(* IEC 61131-3 sources: Industry-PLC-LLM/data/PLCBEAD_repo/PLCBEAD_PLCEmbed-main/PLC-BEAD/Source/GEB/HYST_3, 1 file *)

(* ---- HYST_3.ST ---- *)
FUNCTION_BLOCK HYST_3_Block

	VAR_INPUT
		IN :	REAL;
		HYST :	REAL;
		VAL1 :	REAL;
		VAL2 :	REAL;
	END_VAR

	VAR_OUTPUT
		Q1 :	BOOL;
		Q2 :	BOOL;
	END_VAR

	VAR
		X :	REAL;
	END_VAR

	X := HYST * 0.5;
	IF IN < VAL1 - X THEN
		Q1 := TRUE;
	ELSIF IN > VAL1 + X THEN
		Q1 := FALSE;
	END_IF;
	IF IN < VAL2 - X THEN
		Q2 := FALSE;
	ELSIF IN > VAL2 + X THEN
		Q2 := TRUE;
	END_IF;

END_FUNCTION_BLOCK

PROGRAM program0
	VAR
		IN :	REAL;
		HYST :	REAL;
		VAL1 :	REAL;
		VAL2 :	REAL;
		Q1 :	BOOL;
		Q2 :	BOOL;
		func_block : HYST_3_Block;
	END_VAR
	func_block.IN := IN;
	func_block.HYST := HYST;
	func_block.VAL1 := VAL1;
	func_block.VAL2 := VAL2;
	func_block();
	Q1  := func_block.Q1;
	Q2  := func_block.Q2;
END_PROGRAM
